FUNCTION_BLOCK FB_Analog_Out
VAR_INPUT
END_VAR
VAR_IN_OUT
	Input1																: REAL;
	Input2																: REAL;
END_VAR
VAR
	Last1																: REAL;
	Last2																: REAL;
END_VAR

// Phase 0 - FB_Analog_Out
// Rev 1.0 - April 3, 2024

IF Input2 <> Last2 THEN
	Last2																:= Input2;
	Input1																:= Input2;
	Last1																:= Input2;
ELSIF Input1 <> Last1 THEN
	Last1																:= Input1;
	Input2																:= Input1;
	Last2																:= Input1;
END_IF

END_FUNCTION_BLOCK

(* stored: Version 1.1.0.1, ProductVersion 3.1.4024.12
   POU FB_Analog_Out: Id {bb6dbcf1-aa6d-4898-8174-f3abdc4398d1}, SpecialFunc None *)
